FUNCTION_BLOCK AUI_TO_AB (* Composite FB for converting AUI (UINT) adapter to AB (BYTE) adapter *)
  (* Standard: 61499-2; Description: Copyright (c) 2026 HR Agrartechnik GmbH This program and the accompanying materials are made available under the terms of the Eclipse Public License 2.0 which is available at https://www.eclipse.org/legal/epl-2.0/ SPDX-License-Identifier: EPL-2.0 *)
  (* Version 1.0, 2026-02-17, Franz Höpfinger, HR Agrartechnik GmbH *)
  PACKAGE adapter::conversion::unidirectional;
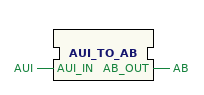
  SOCKETS
    AUI_IN : adapter::types::unidirectional::AUI; (* UINT Adapter Input *)
  END_SOCKETS
  PLUGS
    AB_OUT : adapter::types::unidirectional::AB; (* BYTE Adapter Output *)
  END_PLUGS
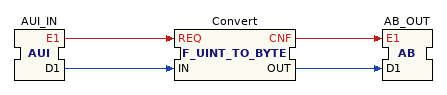
  FBS
    Convert : iec61131::conversion::F_UINT_TO_BYTE;
  END_FBS
  EVENT_CONNECTIONS
    AUI_IN.E1 TO Convert.REQ;
    Convert.CNF TO AB_OUT.E1;
  END_CONNECTIONS
  DATA_CONNECTIONS
    AUI_IN.D1 TO Convert.IN;
    Convert.OUT TO AB_OUT.D1;
  END_CONNECTIONS
END_FUNCTION_BLOCK
